SYSTEM System (* System Configuration *)
  (* Standard: 61499-1 *)
  (* Version 0.0, 1/9/2024, Cheyan, Schneider Electric *)
  {SET_ATTRIBUTE(System.Device.FolderPath, EcoRT_0)}
  APPLICATION APP1
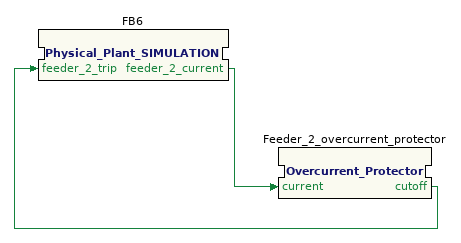
    (* Plant (Power System) *)
    (* Feeder 2 *)
    FBS
      FB6 : Physical_Plant_SIMULATION;
      Feeder_2_overcurrent_protector : Overcurrent_Protector;
    END_FBS
    ADAPTER_CONNECTIONS
      FB6.feeder_2_current TO Feeder_2_overcurrent_protector.current;
      Feeder_2_overcurrent_protector.cutoff TO FB6.feeder_2_trip;
    END_CONNECTIONS
  END_APPLICATION
  DEVICE EcoRT_0 : Soft_dPAC
    RESOURCE RES0 : EMB_RES_ECO
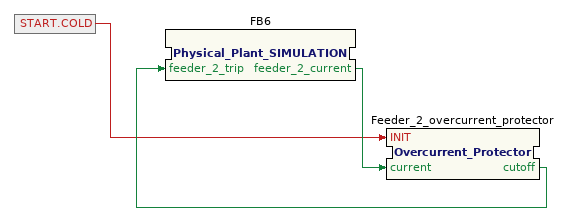
      FBS
        FB6 : Physical_Plant_SIMULATION;
        Feeder_2_overcurrent_protector : Overcurrent_Protector;
      END_FBS
      EVENT_CONNECTIONS
        START.COLD TO Feeder_2_overcurrent_protector.INIT;
      END_CONNECTIONS
      ADAPTER_CONNECTIONS
        FB6.feeder_2_current TO Feeder_2_overcurrent_protector.current;
        Feeder_2_overcurrent_protector.cutoff TO FB6.feeder_2_trip;
      END_CONNECTIONS
    END_RESOURCE
  END_DEVICE
  MAPPINGS
    APP1.FB6 ON EcoRT_0.RES0;
    APP1.Feeder_2_overcurrent_protector ON EcoRT_0.RES0;
  END_MAPPINGS
END_SYSTEM
